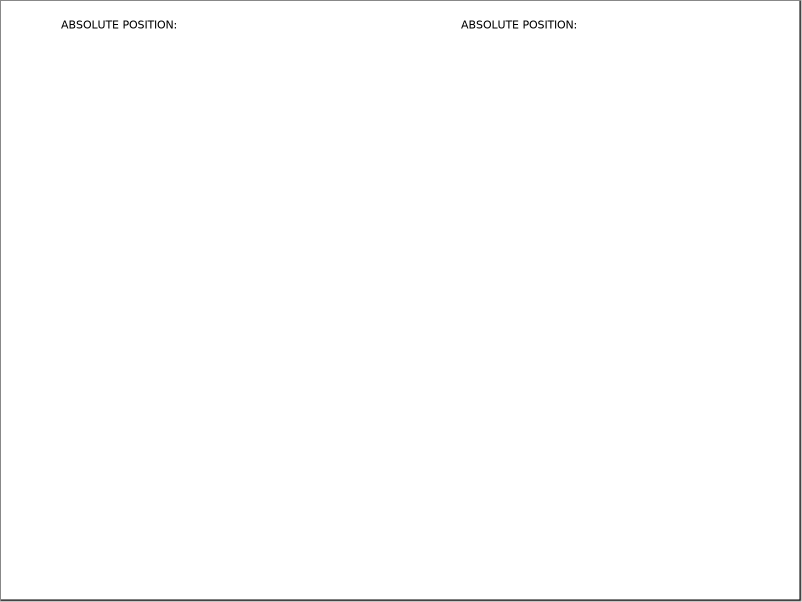
VISUALIZATION F08_Write_Bool_Parameter  // 802x602
    Rectangle (0,0 800x600)
    Label (10,10 170x30), "ABSOLUTE POSITION:"
    Label (410,10 170x30), "ABSOLUTE POSITION:"
END_VISUALIZATION

(* stored: Version 1.1.0.1, ProductVersion 3.1.4022.7
   Visu F08_Write_Bool_Parameter: Id {225a5cf5-5de1-4df8-9eed-d0a8bcb76bcd} *)
